FUNCTION_BLOCK ScaleDecorator IMPLEMENTS ITF_Analogue
VAR
	wrappee : ITF_Analogue;
END_VAR

METHOD GetValue : INT
IF (THIS^.wrappee <> 0) THEN
  GetValue := THIS^.wrappee.GetValue() + 0.9;
END_IF
END_METHOD

END_FUNCTION_BLOCK

(* stored: Version 1.1.0.1, ProductVersion 3.1.4024.12
   POU ScaleDecorator: Id {9cf9a9ee-882f-4ed8-9106-b173b56b8405}, SpecialFunc None
   Method GetValue: Id {23c4be5e-6b38-43f6-adef-2b3982100275} *)
